SUBAPPLICATION Uebung_009 (* Ticker *)
  (* Standard: 61499-2; Description: Copyright (c) 2023 Meisterschulen am Ostbahnhof This program and the accompanying materials are made available under the terms of the Eclipse Public License 2.0 which is available at https://www.eclipse.org/legal/epl-2.0/ SPDX-License-Identifier: EPL-2.0 *)
  (* Version 1.0, 2023-10-23, Franz Höpfinger, Meisterschulen am Ostbahnhof *)
  PACKAGE Uebungen;
  IMPORT Uebungen::const::UT::DefaultPool::OutputNumber_N1;
  IMPORT logiBUS::io::DQ::logiBUS_DO::Output_Q1;
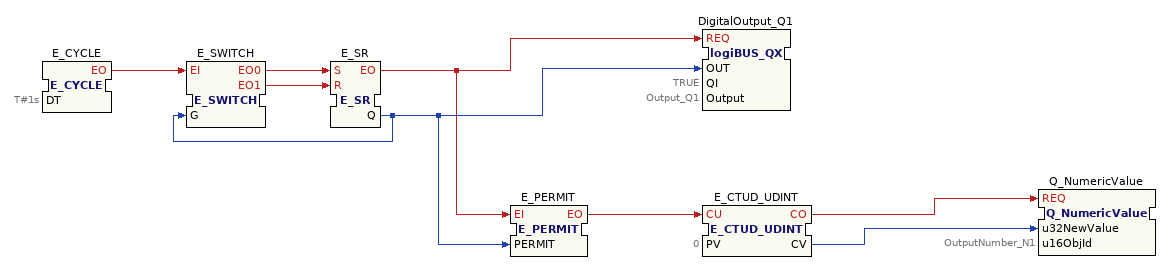
  (* In Watch wechseln, und bei START ein Event auslösen. *)
  FBS
    DigitalOutput_Q1 : logiBUS::io::DQ::logiBUS_QX(QI := TRUE, Output := Output_Q1);
    E_CYCLE : iec61499::events::E_CYCLE(DT := T#1s);
    E_SWITCH : iec61499::events::E_SWITCH;
    E_SR : iec61499::events::E_SR;
    E_PERMIT : iec61499::events::E_PERMIT;
    E_CTUD_UDINT : iec61499::events::E_CTUD_UDINT(PV := 0);
    Q_NumericValue : isobus::UT::Q::Q_NumericValue(u16ObjId := OutputNumber_N1);
  END_FBS
  EVENT_CONNECTIONS
    E_CYCLE.EO TO E_SWITCH.EI;
    E_SWITCH.EO0 TO E_SR.S;
    E_SWITCH.EO1 TO E_SR.R;
    E_SR.EO TO DigitalOutput_Q1.REQ;
    E_SR.EO TO E_PERMIT.EI;
    E_PERMIT.EO TO E_CTUD_UDINT.CU;
    E_CTUD_UDINT.CO TO Q_NumericValue.REQ;
  END_CONNECTIONS
  DATA_CONNECTIONS
    E_SR.Q TO E_SWITCH.G;
    E_SR.Q TO DigitalOutput_Q1.OUT;
    E_SR.Q TO E_PERMIT.PERMIT;
    E_CTUD_UDINT.CV TO Q_NumericValue.u32NewValue;
  END_CONNECTIONS
END_SUBAPPLICATION
